# EPICS autosave request: BPMApp/Db/BPMFmc250m_4ch_settings.req
$(P)$(R)ADC$(ADC_CHAN)TestMode-SP
$(P)$(R)ADC$(ADC_CHAN)RstModes-Sel
